# EPICS substitutions: iocBoot/iocTomoStream_832/tomoStream.substitutions
file "$(TOP)/db/tomoStream.template"
{
pattern
{  P,      R, TOMO_SCAN, IMAGE_P, DARK_PVA, FLAT_PVA, RECON_PVA, THETA_PVA}
{ALS832:, TomoStream:, 7bmtomo:TomoScanStream:, 7bmtomo:TSS:PvaPluginPVPrefix, 7bmtomo:TSS:StreamDarkFields, 7bmtomo:TSS:StreamFlatFields, 7bmtomo:TomoStream:StreamRecon, 7bmtomo:TSS:StreamTheta}
}
